{attribute 'GeneratedUsingTerminal: EL5021-0000-0016'}
{attribute addProperty BoxType "EL5021-0000-0016"}
{attribute addProperty Id "StatusAT %I*Status_A9D949758Counter_valueAT %I*UDINT4Latch_valueAT %I*UDINT4"}
{attribute addProperty CRC "505836508"}
{attribute addProperty Size "16"}
TYPE ENC_Status_1E2673DC EXTENDS InputBase_8311D824 :
STRUCT
	{attribute addProperty Name "Status"}
	Status AT %I* : Status_A9D94975;
	{attribute addProperty Name "Counter_value"}
	Counter_value AT %I* : UDINT;
	{attribute addProperty Name "Latch_value"}
	Latch_value AT %I* : UDINT;
END_STRUCT
END_TYPE

(* stored: Version 1.2.0.0, ProductVersion 3.1.4024.11
   DUT ENC_Status_1E2673DC: Id {6e7881bb-3274-418d-9c04-7afe4c8cca28} *)
